// TIA Portal V20 export
DATA_BLOCK "MotionNodes"   // DB39
// stored: Access Published, MemoryReserve 100, Namespace Unit1
   VAR
      MotionToPLC : "LER_typeMotionToPLC";
      PLCToMotion : "LER_typePLCToMotion";
   END_VAR
BEGIN
   PLCToMotion.TechnologyObject.OutputCam.FinalRollerXFwdOutputCam := 225;
END_DATA_BLOCK
